Omron Sysmac Studio project Benim_Fonk (Sysmac Studio 1.65.0.64007, StandardProject)

# Controller new_Controller_0: NX1P2-1040DT1 version 1.69
Task PrimaryTask (priority 4, period or condition 2000): Program0

VAR_GLOBAL
    AI_Value2 : REAL;
    OnOff : BOOL;
END_VAR

PROGRAM Program0
VAR
    Scale_Value : REAL;
    Scale_X0 : REAL;
    Scale_Y0 : REAL;
    Scale_X1 : REAL;
    Scale_Y1 : REAL;
    Scale_Out : REAL;
    Lim_Min : REAL;
    Lim_Max : REAL;
    Lim_Out : REAL;
    Analog_Input : REAL;
    InputMin : REAL;
    OutputMin : REAL;
    OutputMax : REAL;
    BasinsDeg : REAL;
    InputMax : REAL;
    BenimFiltre_5liOrt : Filtreleme;
    Ton_Pulse : TON;
    Pulse_200ms : BOOL;
    Ortalama_Deger : REAL;
    OnOff : BOOL;
END_VAR
VAR_EXTERNAL
    AI_Value2 : REAL;
END_VAR
VAR
    _t1 : BOOL;
    _p2 : BOOL;
END_VAR

(* Section Section0: ladder, written here as Structured Text *)

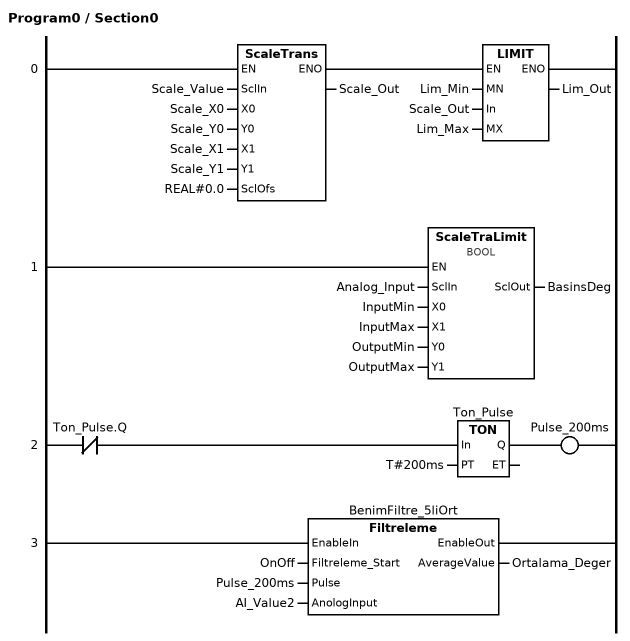
(* Rung 0 *)
Scale_Out := ScaleTrans(SclIn := Scale_Value, X0 := Scale_X0, Y0 := Scale_Y0, X1 := Scale_X1, Y1 := Scale_Y1, SclOfs := REAL#0.0);
Lim_Out := LIMIT(MN := Lim_Min, In := Scale_Out, MX := Lim_Max);
(* Rung 1 *)
_t1 := ScaleTraLimit(SclIn := Analog_Input, X0 := InputMin, X1 := InputMax, Y0 := OutputMin, Y1 := OutputMax, SclOut => BasinsDeg);
(* Rung 2 *)
_p2 := NOT Ton_Pulse.Q;
Ton_Pulse(In := _p2, PT := T#200ms);
Pulse_200ms := Ton_Pulse.Q;
(* Rung 3 *)
BenimFiltre_5liOrt(EnableIn := TRUE, Filtreleme_Start := OnOff, Pulse := Pulse_200ms, AnologInput := AI_Value2, AverageValue => Ortalama_Deger);
END_PROGRAM

FUNCTION ScaleTraLimit : BOOL
VAR
    Scl_Out_Temp : REAL;
END_VAR
VAR_INPUT
    SclIn : REAL;
    X0 : REAL;
    X1 : REAL;
    Y0 : REAL;
    Y1 : REAL;
END_VAR
VAR_OUTPUT
    SclOut : REAL;
END_VAR
(* ladder, written here as Structured Text *)

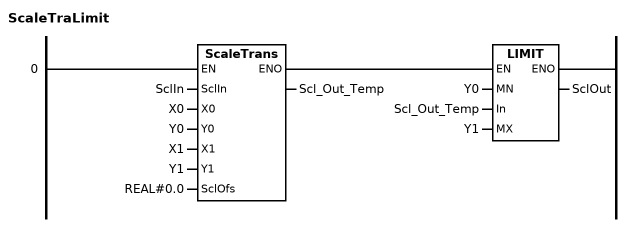
(* Rung 0 *)
Scl_Out_Temp := ScaleTrans(SclIn := SclIn, X0 := X0, Y0 := Y0, X1 := X1, Y1 := Y1, SclOfs := REAL#0.0);
SclOut := LIMIT(MN := Y0, In := Scl_Out_Temp, MX := Y1);
END_FUNCTION

FUNCTION_BLOCK Filtreleme
VAR
    Sayici : INT;
    AnologArry : ARRAY[1..5] OF REAL;
END_VAR
VAR_INPUT
    EnableIn : BOOL;
END_VAR
VAR_OUTPUT
    EnableOut : BOOL;
END_VAR
VAR_INPUT
    Filtreleme_Start : BOOL;
    Pulse : BOOL;
    AnologInput : REAL;
END_VAR
VAR_OUTPUT
    AverageValue : REAL;
END_VAR
VAR
    _e1 : R_TRIG;
    _e2 : R_TRIG;
    _e3 : R_TRIG;
    _e4 : R_TRIG;
    _e5 : R_TRIG;
    _e6 : R_TRIG;
    _e7 : R_TRIG;
END_VAR
(* ladder, written here as Structured Text *)

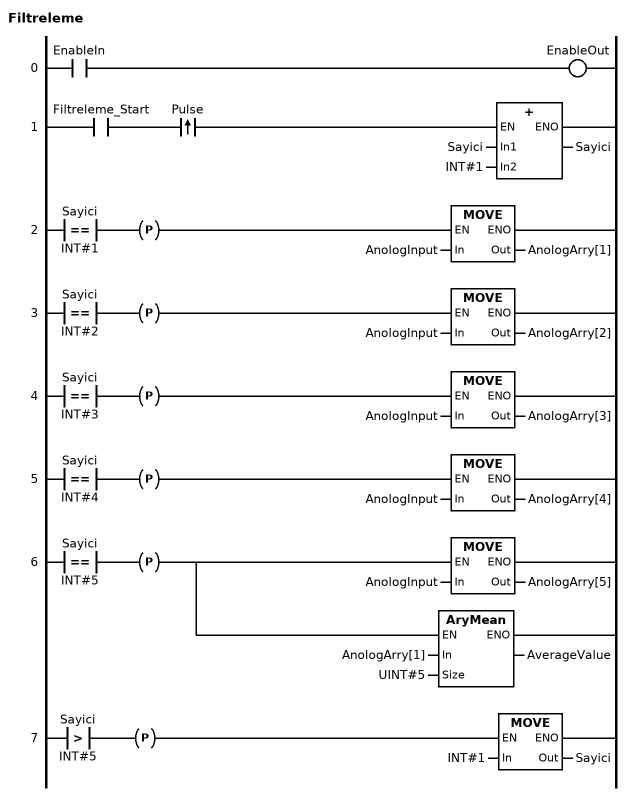
(* Rung 0 *)
EnableOut := EnableIn;
(* Rung 1 *)
_e1(CLK := Pulse);
IF Filtreleme_Start AND _e1.Q THEN Sayici := Sayici + INT#1; END_IF;
(* Rung 2 *)
_e2(CLK := Sayici = INT#1);
IF _e2.Q THEN AnologArry[1] := AnologInput; END_IF;
(* Rung 3 *)
_e3(CLK := Sayici = INT#2);
IF _e3.Q THEN AnologArry[2] := AnologInput; END_IF;
(* Rung 4 *)
_e4(CLK := Sayici = INT#3);
IF _e4.Q THEN AnologArry[3] := AnologInput; END_IF;
(* Rung 5 *)
_e5(CLK := Sayici = INT#4);
IF _e5.Q THEN AnologArry[4] := AnologInput; END_IF;
(* Rung 6 *)
_e6(CLK := Sayici = INT#5);
IF _e6.Q THEN
    AnologArry[5] := AnologInput;
    AverageValue := AryMean(In := AnologArry[1], Size := UINT#5);
END_IF;
(* Rung 7 *)
_e7(CLK := Sayici > INT#5);
IF _e7.Q THEN Sayici := INT#1; END_IF;
END_FUNCTION_BLOCK